// TIA Portal V20 export
TYPE "typeSequenceControlNode"
// stored: Namespace Unit1.Em10
   STRUCT
      jobs : "LAF_typeJobs";
      sequence : "LAF_typeSequence";
      selectJobStatus { S7_SetPoint := 'True'} : Array[0..10] of "LAF_typeJobStatus";
      "step" : "LER_typeStep";
      jobInterface : "Unit1.Em10.typeSequenceControlNodeJobInterface";
      homeCheck : "Unit1.Em10.typeSequenceControlNodeHomeCheck";
   END_STRUCT;
   // // "step".action1[101] : Step[101] : JOB[1] Condition
   // // "step".action1[130] : Step[130] : Stage Lift Up
   // // "step".action1[140] : Step[140] : Hot Press Left JR Detection Check
   // // "step".action1[141] : Step[141] : Hot Press Left JR Detection Check Completed
   // // "step".action1[160] : Step[160] : Stage Lift Down, Cover Up
   // // "step".action1[190] : Step[190] : JOB[1] Step End
   // // "step".action1[201] : Step[201] : JOB[2] Condition
   // // "step".action1[210] : Step[210] : Laser Mark Loading Request => Transfer PP Right
   // // "step".action1[230] : Step[230] : Stage Lift Up
   // // "step".action1[240] : Step[240] : Laser Mark Loading Check => Transfer PP Right
   // // "step".action1[250] : Step[250] : Laser Mark JR Detection Check
   // // "step".action1[290] : Step[290] : JOB[2] Step End
   // // "step".action1[301] : Step[301] : JOB[3] Condition
   // // "step".action1[310] : Step[310] : Stage Lift, Cover Down
   // // "step".action1[311] : Step[311] : Stage Lift, Cover Down
   // // "step".action1[330] : Step[330] : Laser Mark Start
   // // "step".action1[331] : Step[331] : Laser Mark Result
   // // "step".action1[340] : Step[340] : NG Data Generate
   // // "step".action1[341] : Step[341] : Laser Mark Start [NG]
   // // "step".action1[342] : Step[342] : Laser Mark Result [NG]
   // // "step".action1[390] : Step[390] : JOB[3] Step End
   // // "step".action1[401] : Step[401] : JOB[4] Condition
   // // "step".action1[410] : Step[410] : Stage Lift, Cover Up
   // // "step".action1[430] : Step[430] : Laser Mark Unloading Request => Transfer PP Right
   // // "step".action1[431] : Step[431] : Laser Mark Unloading Check => Transfer PP Right
   // // "step".action1[480] : Step[480] : Stage Lift Down
   // // "step".action1[490] : Step[490] : JOB[4] Step End
   // // "step".transition1[101] : Step[101] : JOB[1] Condition
   // // "step".transition1[130] : Step[130] : Stage Lift Up
   // // "step".transition1[140] : Step[140] : Hot Press Left JR Detection Check
   // // "step".transition1[141] : Step[141] : Hot Press Left JR Detection Check Completed
   // // "step".transition1[160] : Step[160] : Stage Lift Down, Cover Up
   // // "step".transition1[190] : Step[190] : JOB[1] Step End
   // // "step".transition1[201] : Step[201] : JOB[2] Condition
   // // "step".transition1[210] : Step[210] : Laser Mark Loading Request => Transfer PP Right
   // // "step".transition1[230] : Step[230] : Stage Lift Up
   // // "step".transition1[240] : Step[240] : Laser Mark Loading Check => Transfer PP Right
   // // "step".transition1[250] : Step[250] : Laser Mark JR Detection Check
   // // "step".transition1[290] : Step[290] : JOB[2] Step End
   // // "step".transition1[301] : Step[301] : JOB[3] Condition
   // // "step".transition1[310] : Step[310] : Stage Lift, Cover Down
   // // "step".transition1[311] : Step[311] : Stage Lift, Cover Down
   // // "step".transition1[330] : Step[330] : Laser Mark Start
   // // "step".transition1[331] : Step[331] : Laser Mark Result
   // // "step".transition1[340] : Step[340] : NG Data Generate
   // // "step".transition1[341] : Step[341] : Laser Mark Start [NG]
   // // "step".transition1[342] : Step[342] : Laser Mark Result [NG]
   // // "step".transition1[390] : Step[390] : JOB[3] Step End
   // // "step".transition1[401] : Step[401] : JOB[4] Condition
   // // "step".transition1[410] : Step[410] : Stage Lift, Cover Up
   // // "step".transition1[430] : Step[430] : Laser Mark Unloading Request => Transfer PP Right
   // // "step".transition1[431] : Step[431] : Laser Mark Unloading Check => Transfer PP Right
   // // "step".transition1[480] : Step[480] : Stage Lift Down
   // // "step".transition1[490] : Step[490] : JOB[4] Step End
END_TYPE
